% RSLogix 500 project Project_7.RSS, saved by version 8.30.00.16 %
PROJECT "UNTITLED"    % processor: Bul.1763 MicroLogix 1100 Series B %

PROGRAM FILES
  LAD 2   3 rungs
  LAD 3 "IO"  3 rungs  % Input/Output %
  LAD 4 "LOGIC"  20 rungs  % Logic %

DATA FILES
  O0 OUTPUT  4 elements
  I1 INPUT  6 elements
  S2 STATUS  66 elements
  B3 BINARY  1 elements
  T4 TIMER  2 elements
  C5 COUNTER  2 elements
  R6 CONTROL  1 elements
  N7 INTEGER  30 elements
  F8 FLOAT  20 elements

LADDER 2
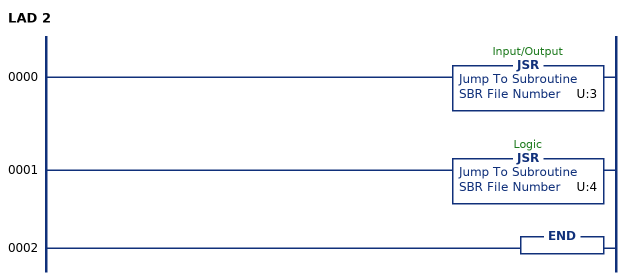
% Rung: 0 %
SOR JSR U:3 EOR
%   U:3  "Input/Output" %
% Rung: 1 %
SOR JSR U:4 EOR
%   U:4  "Logic" %
% Rung: 2 %
SOR END EOR

LADDER 3 "IO"    % Input/Output %
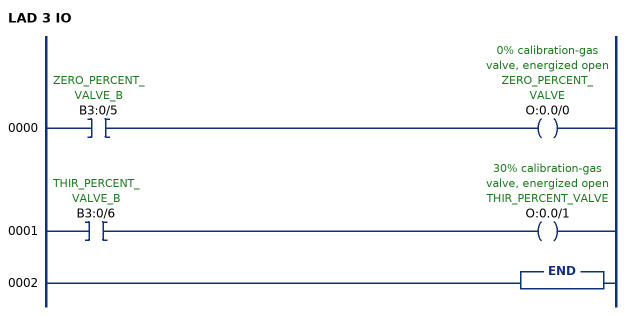
% Rung: 0 %
SOR XIC B3:0/5 OTE O:0.0/0 EOR
%   B3:0/5  ZERO_PERCENT_VALVE_B %
%   O:0.0/0  ZERO_PERCENT_VALVE  "0% calibration-gas valve, energized open" %
% Rung: 1 %
SOR XIC B3:0/6 OTE O:0.0/1 EOR
%   B3:0/6  THIR_PERCENT_VALVE_B %
%   O:0.0/1  THIR_PERCENT_VALVE  "30% calibration-gas valve, energized open" %
% Rung: 2 %
SOR END EOR

LADDER 4 "LOGIC"    % Logic %
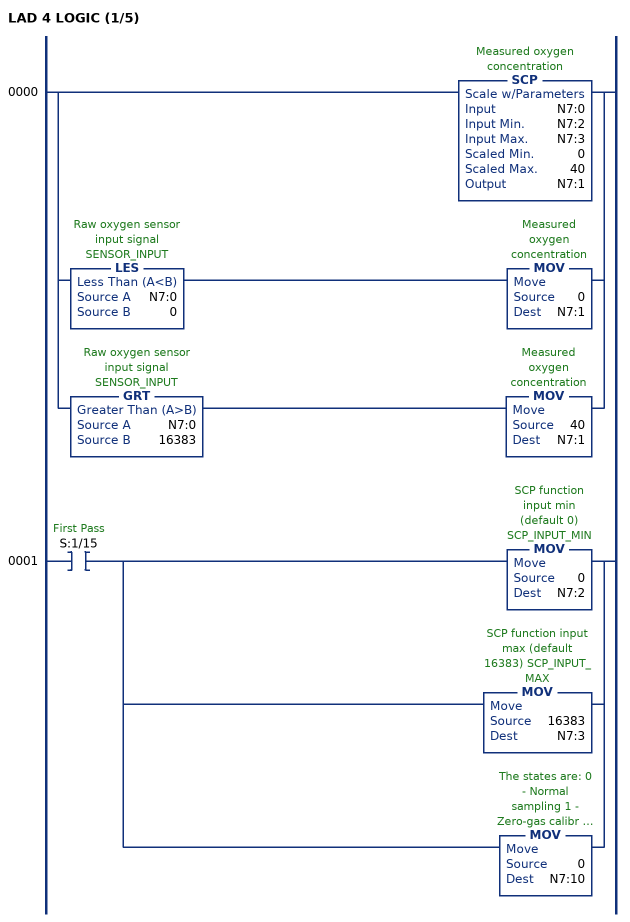
% Rung: 0 %
SOR BST SCP N7:0 N7:2 N7:3 0 40 N7:1 NXB BST LES N7:0 0 MOV 0 N7:1 NXB GRT N7:0 16383 MOV 40 N7:1 BND BND EOR
%   N7:0  SENSOR_INPUT  "Raw oxygen sensor input signal" %
%   N7:2  SCP_INPUT_MIN  "SCP function input min (default 0)" %
%   N7:3  SCP_INPUT_MAX  "SCP function input max (default 16383)" %
%   N7:1  "Measured oxygen concentration" %
% Rung: 1 %
SOR XIC S:1/15 BST MOV 0 N7:2 NXB BST MOV 16383 N7:3 NXB MOV 0 N7:10 BND BND EOR
%   S:1/15  "First Pass" %
%   N7:2  SCP_INPUT_MIN  "SCP function input min (default 0)" %
%   N7:3  SCP_INPUT_MAX  "SCP function input max (default 16383)" %
%   N7:10  STATE  "The states are: 0 - Normal sampling 1 - Zero-gas calibr 2 - 30% gas calibr 3 - Calc and apply" %

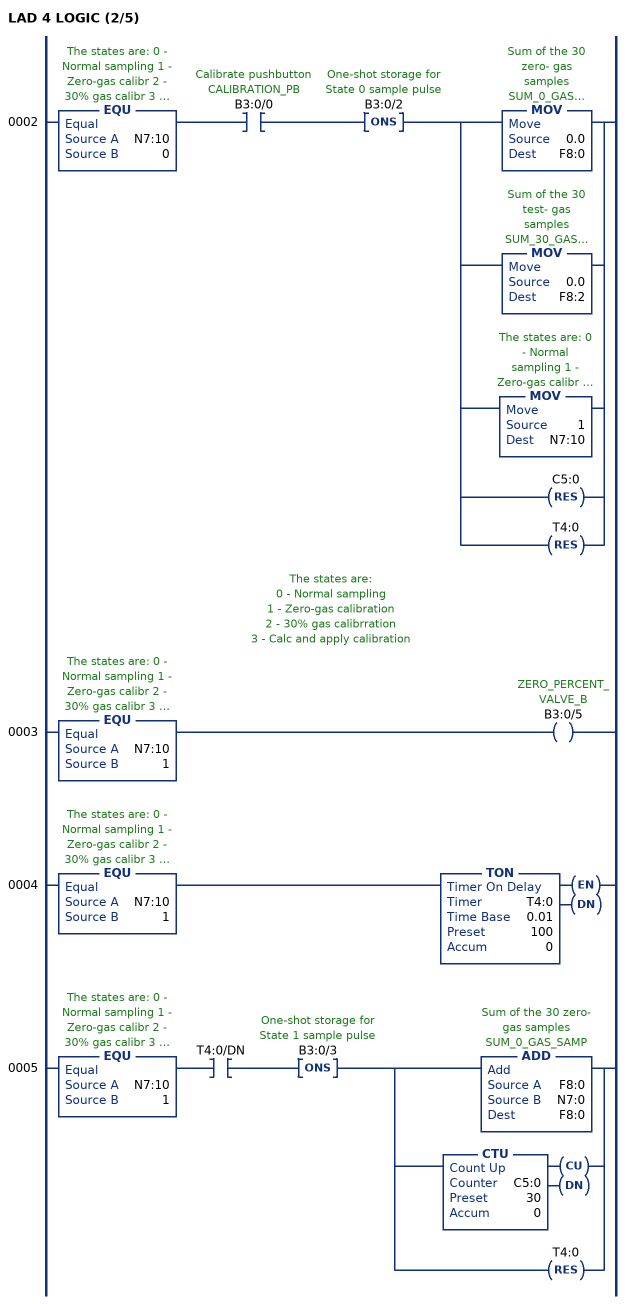
% Rung: 2 %
SOR EQU N7:10 0 XIC B3:0/0 ONS B3:0/2 BST MOV 0.0 F8:0 NXB BST MOV 0.0 F8:2 NXB BST MOV 1 N7:10 NXB BST RES C5:0 NXB RES T4:0 BND BND BND BND EOR
%   N7:10  STATE  "The states are: 0 - Normal sampling 1 - Zero-gas calibr 2 - 30% gas calibr 3 - Calc and apply" %
%   B3:0/0  CALIBRATION_PB  "Calibrate pushbutton" %
%   B3:0/2  "One-shot storage for State 0 sample pulse" %
%   F8:0  SUM_0_GAS_SAMP  "Sum of the 30 zero- gas samples" %
%   F8:2  SUM_30_GAS_SAMP  "Sum of the 30 test- gas samples" %
% Rung: 3 %
% The states are:
% 0 - Normal sampling
% 1 - Zero-gas calibration
% 2 - 30% gas calibrration
% 3 - Calc and apply calibration %
SOR EQU N7:10 1 OTE B3:0/5 EOR
%   N7:10  STATE  "The states are: 0 - Normal sampling 1 - Zero-gas calibr 2 - 30% gas calibr 3 - Calc and apply" %
%   B3:0/5  ZERO_PERCENT_VALVE_B %
% Rung: 4 %
SOR EQU N7:10 1 TON T4:0 0.01 100 0 EOR
%   N7:10  STATE  "The states are: 0 - Normal sampling 1 - Zero-gas calibr 2 - 30% gas calibr 3 - Calc and apply" %
% Rung: 5 %
SOR EQU N7:10 1 XIC T4:0/DN ONS B3:0/3 BST ADD F8:0 N7:0 F8:0 NXB BST CTU C5:0 30 0 NXB RES T4:0 BND BND EOR
%   N7:10  STATE  "The states are: 0 - Normal sampling 1 - Zero-gas calibr 2 - 30% gas calibr 3 - Calc and apply" %
%   B3:0/3  "One-shot storage for State 1 sample pulse" %
%   F8:0  SUM_0_GAS_SAMP  "Sum of the 30 zero- gas samples" %
%   N7:0  SENSOR_INPUT  "Raw oxygen sensor input signal" %

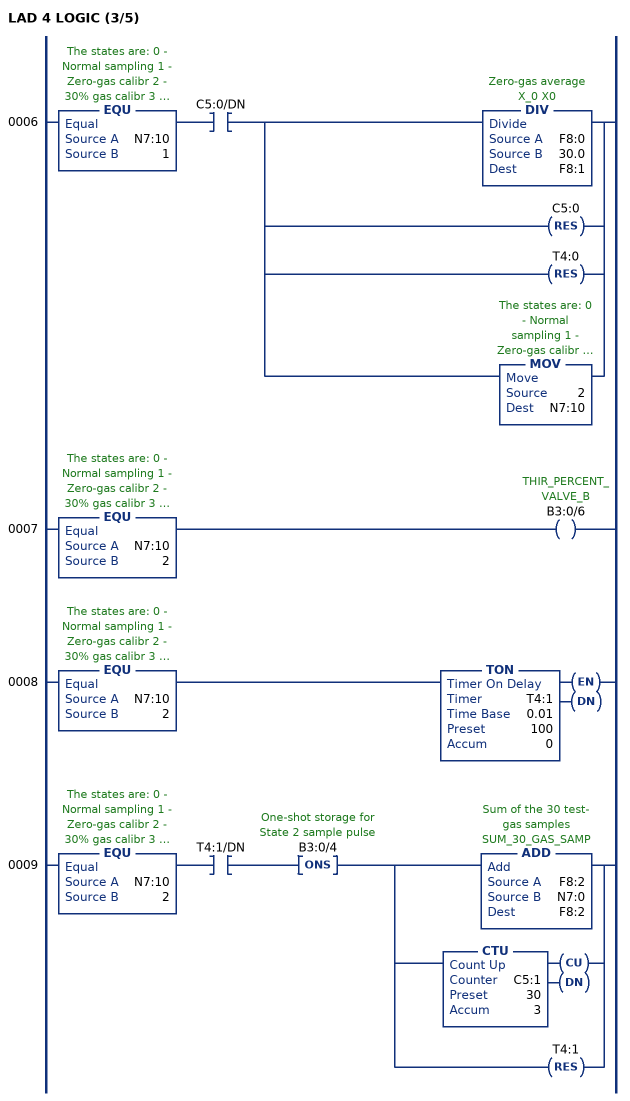
% Rung: 6 %
SOR EQU N7:10 1 XIC C5:0/DN BST DIV F8:0 30.0 F8:1 NXB BST RES C5:0 NXB BST RES T4:0 NXB MOV 2 N7:10 BND BND BND EOR
%   N7:10  STATE  "The states are: 0 - Normal sampling 1 - Zero-gas calibr 2 - 30% gas calibr 3 - Calc and apply" %
%   F8:0  SUM_0_GAS_SAMP  "Sum of the 30 zero- gas samples" %
%   F8:1  X0  "Zero-gas average X_0" %
% Rung: 7 %
SOR EQU N7:10 2 OTE B3:0/6 EOR
%   N7:10  STATE  "The states are: 0 - Normal sampling 1 - Zero-gas calibr 2 - 30% gas calibr 3 - Calc and apply" %
%   B3:0/6  THIR_PERCENT_VALVE_B %
% Rung: 8 %
SOR EQU N7:10 2 TON T4:1 0.01 100 0 EOR
%   N7:10  STATE  "The states are: 0 - Normal sampling 1 - Zero-gas calibr 2 - 30% gas calibr 3 - Calc and apply" %
% Rung: 9 %
SOR EQU N7:10 2 XIC T4:1/DN ONS B3:0/4 BST ADD F8:2 N7:0 F8:2 NXB BST CTU C5:1 30 3 NXB RES T4:1 BND BND EOR
%   N7:10  STATE  "The states are: 0 - Normal sampling 1 - Zero-gas calibr 2 - 30% gas calibr 3 - Calc and apply" %
%   B3:0/4  "One-shot storage for State 2 sample pulse" %
%   F8:2  SUM_30_GAS_SAMP  "Sum of the 30 test- gas samples" %
%   N7:0  SENSOR_INPUT  "Raw oxygen sensor input signal" %

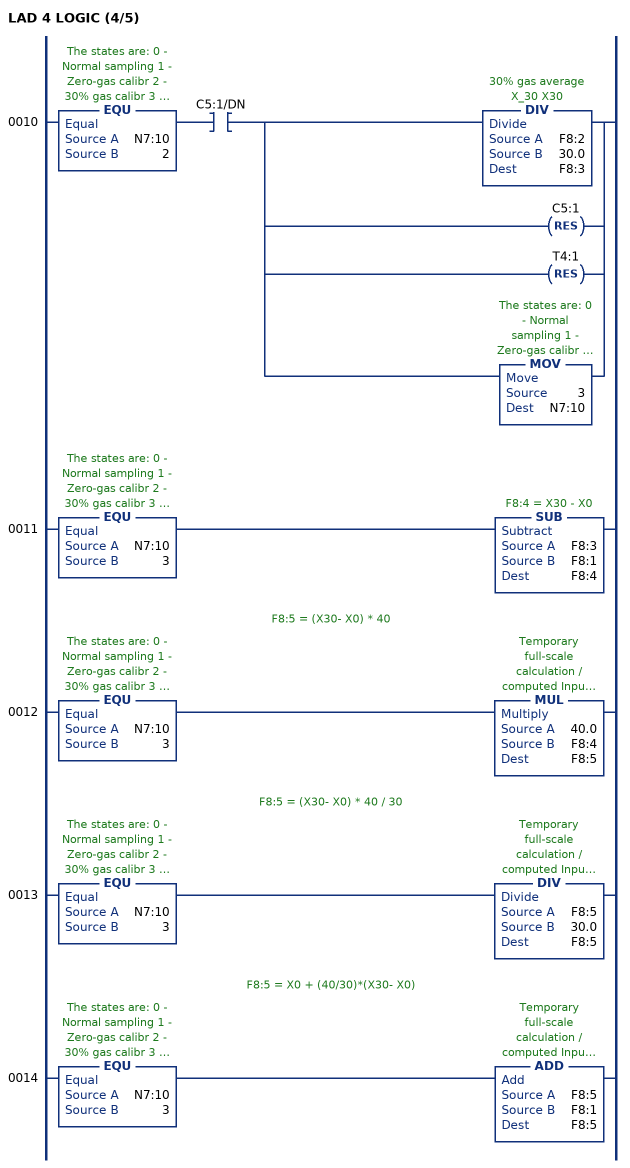
% Rung: 10 %
SOR EQU N7:10 2 XIC C5:1/DN BST DIV F8:2 30.0 F8:3 NXB BST RES C5:1 NXB BST RES T4:1 NXB MOV 3 N7:10 BND BND BND EOR
%   N7:10  STATE  "The states are: 0 - Normal sampling 1 - Zero-gas calibr 2 - 30% gas calibr 3 - Calc and apply" %
%   F8:2  SUM_30_GAS_SAMP  "Sum of the 30 test- gas samples" %
%   F8:3  X30  "30% gas average X_30" %
% Rung: 11 %
SOR EQU N7:10 3 SUB F8:3 F8:1 F8:4 EOR
%   N7:10  STATE  "The states are: 0 - Normal sampling 1 - Zero-gas calibr 2 - 30% gas calibr 3 - Calc and apply" %
%   F8:3  X30  "30% gas average X_30" %
%   F8:1  X0  "Zero-gas average X_0" %
%   F8:4  "F8:4 = X30 - X0" %
% Rung: 12 %
%  F8:5 = (X30- X0) * 40 %
SOR EQU N7:10 3 MUL 40.0 F8:4 F8:5 EOR
%   N7:10  STATE  "The states are: 0 - Normal sampling 1 - Zero-gas calibr 2 - 30% gas calibr 3 - Calc and apply" %
%   F8:4  "F8:4 = X30 - X0" %
%   F8:5  "Temporary full-scale calculation / computed Input Max" %
% Rung: 13 %
%  F8:5 = (X30- X0) * 40 / 30 %
SOR EQU N7:10 3 DIV F8:5 30.0 F8:5 EOR
%   N7:10  STATE  "The states are: 0 - Normal sampling 1 - Zero-gas calibr 2 - 30% gas calibr 3 - Calc and apply" %
%   F8:5  "Temporary full-scale calculation / computed Input Max" %
% Rung: 14 %
% F8:5 = X0 + (40/30)*(X30- X0) %
SOR EQU N7:10 3 ADD F8:5 F8:1 F8:5 EOR
%   N7:10  STATE  "The states are: 0 - Normal sampling 1 - Zero-gas calibr 2 - 30% gas calibr 3 - Calc and apply" %
%   F8:5  "Temporary full-scale calculation / computed Input Max" %
%   F8:1  X0  "Zero-gas average X_0" %

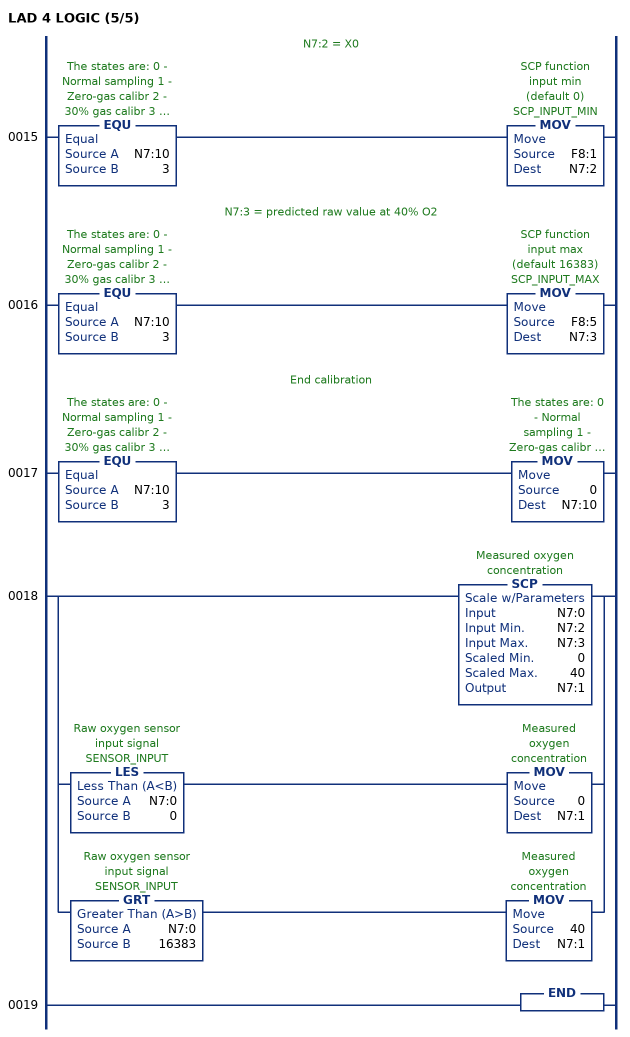
% Rung: 15 %
%  N7:2 = X0 %
SOR EQU N7:10 3 MOV F8:1 N7:2 EOR
%   N7:10  STATE  "The states are: 0 - Normal sampling 1 - Zero-gas calibr 2 - 30% gas calibr 3 - Calc and apply" %
%   F8:1  X0  "Zero-gas average X_0" %
%   N7:2  SCP_INPUT_MIN  "SCP function input min (default 0)" %
% Rung: 16 %
% N7:3 = predicted raw value at 40% O2 %
SOR EQU N7:10 3 MOV F8:5 N7:3 EOR
%   N7:10  STATE  "The states are: 0 - Normal sampling 1 - Zero-gas calibr 2 - 30% gas calibr 3 - Calc and apply" %
%   F8:5  "Temporary full-scale calculation / computed Input Max" %
%   N7:3  SCP_INPUT_MAX  "SCP function input max (default 16383)" %
% Rung: 17 %
% End calibration %
SOR EQU N7:10 3 MOV 0 N7:10 EOR
%   N7:10  STATE  "The states are: 0 - Normal sampling 1 - Zero-gas calibr 2 - 30% gas calibr 3 - Calc and apply" %
% Rung: 18 %
SOR BST SCP N7:0 N7:2 N7:3 0 40 N7:1 NXB BST LES N7:0 0 MOV 0 N7:1 NXB GRT N7:0 16383 MOV 40 N7:1 BND BND EOR
%   N7:0  SENSOR_INPUT  "Raw oxygen sensor input signal" %
%   N7:2  SCP_INPUT_MIN  "SCP function input min (default 0)" %
%   N7:3  SCP_INPUT_MAX  "SCP function input max (default 16383)" %
%   N7:1  "Measured oxygen concentration" %
% Rung: 19 %
SOR END EOR

COMMENTS NOT ATTACHED TO A CURRENT RUNG
  N7:0: Quickly move 8192 to N7:0 to simulate 0% raw measurement

DATA TABLE (non-zero values as saved)
DATA B3
% B3:0 % 0X0041
DATA T4
% .PRE .ACC %
% T4:0 % 100 0
% T4:1 % 100 0
DATA C5
% .PRE .ACC %
% C5:0 % 30 0
% C5:1 % 30 3
DATA N7
% N7:0 % 8192 30 0 16383 0 0 0 0 0 0
% N7:10 % 2 0 0 0 0 0 0 0 0 0
DATA F8
% F8:0 % 245760 8192 36864 12288 4096
% F8:5 % 13653.33 0 0 0 0
